// TwinCAT 3 PLC project PLC_UED_SDS
// ProgramVersion: 3.1.4023.0
// libraries:
//   LCLS General, * (SLAC)
//   LCLS Vacuum, * (SLAC - LCLS)
//   lcls-twincat-sample-delivery, * (SLAC)
//   Tc2_Standard, * (Beckhoff Automation GmbH)
//   Tc2_System, * (Beckhoff Automation GmbH)
//   Tc3_Module, * (Beckhoff Automation GmbH)
// project tree:
//   / PlcTask.TcTTO
//   POUs/ MAIN.TcPOU, PRG_RCC.TcPOU
// real-time tasks:
//   TASK PlcTask: cycle T#10ms, priority 20, ADS port 350
// I/O:
//   DEVICE Device 1 (EtherCAT), AmsNetId 172.21.36.53.2.1
//     Term 1 (EK1200) [EK1200-5000 EtherCAT Power supply (2A E-Bus)]
//       RCC_E1 (EL2004)
//       RCC_E2 (EL1004) [EL1004 4Ch. Dig. Input 24V, 3ms]
//       RCC_E3 (EL1004) [EL1004 4Ch. Dig. Input 24V, 3ms]
//       RCC_TC (EL3314) [EL3314 4Ch. Ana. Input Thermocouple (TC)]
//       Term 6 (EK1110) [EK1110 EtherCAT extension]
//     Box 18 (EP9128-0021) [EP9128-0021 8x EtherCAT junction]
//       BR (EP1111-0000) [EP1111-0000 ID-Switch]
//       BR Valves (EP2338-0001) [EP2338-0001 8 Ch. Dig. Input/Output 24V, 0,5A, M8]
//       Term 23 (EP9128-1021) [EP9128-1021 8x EtherCAT junction - Dev A]
//       Term 24 (EP9128-2021) [EP9128-2021 8x EtherCAT junction - Dev B]
//         Box 25 (EP1111) [EP1111-0000 ID-Switch]
//         Box 26 (EP2338-0001) [EP2338-0001 8 Ch. Dig. Input/Output 24V, 0,5A, M8]
//         4PortVICI Serial (EP6002-0002) [EP6002-0002 Interface (RS232/422/485)]
// variable links:
//   PLC_UED_SDS Instance <-> Device 1 (EtherCAT)/Box 18 (EP9128-0021)/BR Valves (EP2338-0001)
//     PlcTask Outputs/MAIN.PURGE_VRC_01_CTL <-> Channel 11/Output
//     PlcTask Outputs/MAIN.PURGE_VRC_02_CTL <-> Channel 12/Output
//     PlcTask Outputs/MAIN.SolenoidPairA.q_xDO1 <-> Channel 9/Output
//     PlcTask Outputs/MAIN.SolenoidPairA.q_xDO2 <-> Channel 10/Output
//   PLC_UED_SDS Instance <-> Device 1 (EtherCAT)/Box 18 (EP9128-0021)/Term 24 (EP9128-2021)/4PortVICI Serial (EP6002-0002)
//     PlcTask Inputs/MAIN.fbValve.fbNporValve.stViciSerial.stComIn/D <-> COM TxPDO-Map Inputs Channel 2/Data In 0
//     PlcTask Inputs/MAIN.fbValve.fbNporValve.stViciSerial.stComIn/D @bit {8..168 step 8} <-> COM TxPDO-Map Inputs Channel 2/Data In {1..21}  (21 links)
//     PlcTask Inputs/MAIN.fbValve.fbNporValve.stViciSerial.stComIn/Status <-> COM TxPDO-Map Inputs Channel 2/Status
//     PlcTask Outputs/MAIN.fbValve.fbNporValve.stViciSerial.stComOut/Ctrl <-> COM RxPDO-Map Outputs Channel 2/Ctrl
//     PlcTask Outputs/MAIN.fbValve.fbNporValve.stViciSerial.stComOut/D <-> COM RxPDO-Map Outputs Channel 2/Data Out 0
//     PlcTask Outputs/MAIN.fbValve.fbNporValve.stViciSerial.stComOut/D @bit {8..168 step 8} <-> COM RxPDO-Map Outputs Channel 2/Data Out {1..21}  (21 links)
//   PLC_UED_SDS Instance <-> Device 1 (EtherCAT)/Term 1 (EK1200)/RCC_E1 (EL2004)
//     PlcTask Outputs/PRG_RCC.RCC_VRC_01.q_xOPN_DO <-> Channel 1/Output
//     PlcTask Outputs/PRG_RCC.RCC_VRC_02.q_xOPN_DO <-> Channel 2/Output
//     PlcTask Outputs/PRG_RCC.RCC_VRC_03.q_xOPN_DO <-> Channel 3/Output
//     PlcTask Outputs/PRG_RCC.RCC_VRC_04.q_xOPN_DO <-> Channel 4/Output
//   PLC_UED_SDS Instance <-> Device 1 (EtherCAT)/Term 1 (EK1200)/RCC_E2 (EL1004)
//     PlcTask Inputs/PRG_RCC.RCC_VRC_01.i_xClsLS <-> Channel 1/Input
//     PlcTask Inputs/PRG_RCC.RCC_VRC_02.i_xClsLS <-> Channel 2/Input
//     PlcTask Inputs/PRG_RCC.RCC_VRC_03.i_xClsLS <-> Channel 3/Input
//     PlcTask Inputs/PRG_RCC.RCC_VRC_04.i_xClsLS <-> Channel 4/Input
//   PLC_UED_SDS Instance <-> Device 1 (EtherCAT)/Term 1 (EK1200)/RCC_GPI (EL3174-0002)
//     PlcTask Inputs/PRG_RCC.RCC_GCP_01.i_iPRESS_R <-> AI Standard Channel 1/Value
//   PLC_UED_SDS Instance <-> Device 1 (EtherCAT)/Term 1 (EK1200)/RCC_TC (EL3314)
//     PlcTask Inputs/PRG_RCC.RCC_STC_01.bError <-> TC Inputs Channel 1/Status/Error
//     PlcTask Inputs/PRG_RCC.RCC_STC_01.bOverrange <-> TC Inputs Channel 1/Status/Overrange
//     PlcTask Inputs/PRG_RCC.RCC_STC_01.bUnderrange <-> TC Inputs Channel 1/Status/Underrange
//     PlcTask Inputs/PRG_RCC.RCC_STC_01.iRaw <-> TC Inputs Channel 1/Value

CONFIGURATION PLC_UED_SDS
    RESOURCE PLC ON TwinCAT3
        TASK PlcTask(INTERVAL := T#10ms, PRIORITY := 20);
        PROGRAM MAIN WITH PlcTask : MAIN;
    END_RESOURCE
END_CONFIGURATION

// ---- POUs/MAIN.TcPOU
PROGRAM MAIN
VAR
    // 4 Port Valve
    {attribute 'pytmc' := 'pv: UED:SDS:VICI:01'}
    {attribute 'TcLinkTo' := '.fbNporValve.stViciSerial.stComIn.Status := TIID^Device 1 (EtherCAT)^Box 18 (EP9128-0021)^Term 24 (EP9128-2021)^4PortVICI Serial (EP6002-0002)^COM TxPDO-Map Inputs Channel 2^Status;
                              .fbNporValve.stViciSerial.stComOut.Ctrl := TIID^Device 1 (EtherCAT)^Box 18 (EP9128-0021)^Term 24 (EP9128-2021)^4PortVICI Serial (EP6002-0002)^COM RxPDO-Map Outputs Channel 2^Ctrl
    '}
    fbValve : FB_4PortViciValve;

    // ON/OFF Valves
    {attribute 'pytmc' := 'pv: UED:SDS:SPR:A'}
    {attribute 'TcLinkTo' := '.q_xDO1 := TIID^Device 1 (EtherCAT)^Box 18 (EP9128-0021)^BR Valves (EP2338-0001)^Channel 9^Output;
                              .q_xDO2 := TIID^Device 1 (EtherCAT)^Box 18 (EP9128-0021)^BR Valves (EP2338-0001)^Channel 10^Output
    '}
    SolenoidPairA : FB_SolenoidPair;

    // Purge Valves
    {attribute 'pytmc' := 'pv: UED:SDS:PURGE:A'}
    {attribute 'TcLinkTo' := 'TIID^Device 1 (EtherCAT)^Box 18 (EP9128-0021)^BR Valves (EP2338-0001)^Channel 11^Output'}
    PURGE_VRC_01_CTL AT%Q* : BOOL;

    {attribute 'pytmc' := 'pv: UED:SDS:PURGE:B'}
    {attribute 'TcLinkTo' := 'TIID^Device 1 (EtherCAT)^Box 18 (EP9128-0021)^BR Valves (EP2338-0001)^Channel 12^Output'}
    PURGE_VRC_02_CTL AT%Q* : BOOL;

END_VAR

PRG_RCC();
SolenoidPairA();
fbValve(iAdress:=1);

END_PROGRAM

// ---- POUs/PRG_RCC.TcPOU
PROGRAM PRG_RCC
VAR
    (* OverrideMode *)
    {attribute 'pytmc' := 'pv: UED:RCC:VAC:OVRD_MODE'}
    xSystemOverrideMode_RCC	: BOOL := FALSE;


    {attribute 'pytmc' :=' pv: UED:RCC:VRC:01 '}
    {attribute 'TcLinkTo' := 	'.i_xClsLS	:=  TIID^Device 1 (EtherCAT)^Term 1 (EK1200)^RCC_E2 (EL1004)^Channel 1^Input;
                                .q_xOPN_DO	:=	TIID^Device 1 (EtherCAT)^Term 1 (EK1200)^RCC_E1 (EL2004)^Channel 1^Output'}
    RCC_VRC_01 : FB_VRC_NC_ClsLS;


    {attribute 'pytmc' :=' pv: UED:RCC:VRC:02 '}
    {attribute 'TcLinkTo' := 	'.i_xClsLS	:=  TIID^Device 1 (EtherCAT)^Term 1 (EK1200)^RCC_E2 (EL1004)^Channel 2^Input;
                                .q_xOPN_DO	:=	TIID^Device 1 (EtherCAT)^Term 1 (EK1200)^RCC_E1 (EL2004)^Channel 2^Output'}
    RCC_VRC_02 : FB_VRC_NC_ClsLS;

    // RIX RCC USES
    //{attribute 'pytmc' :=' pv: UED:RCC:VRC:02 '}
    //{attribute 'TcLinkTo' := 	'.i_xOpnLS	:= 	TIID^Device 1 (EtherCAT)^Term 1 (EK1200)^RCC_E2 (EL1004)^Channel 3^Input;
    //                             .i_xClsLS	:=	TIID^Device 1 (EtherCAT)^Term 1 (EK1200)^RCC_E2 (EL1004)^Channel 4^Input;
    //                            .q_xOPN_DO	:=	TIID^Device 1 (EtherCAT)^Term 1 (EK1200)^RCC_E1 (EL2004)^Channel 2^Output'}
    //RCC_VRC_02 : FB_VRC;

    {attribute 'pytmc' :=' pv: UED:RCC:VRC:03 '}
    {attribute 'TcLinkTo' := 	'.i_xClsLS	:=	TIID^Device 1 (EtherCAT)^Term 1 (EK1200)^RCC_E2 (EL1004)^Channel 3^Input;
                                .q_xOPN_DO	:= 	TIID^Device 1 (EtherCAT)^Term 1 (EK1200)^RCC_E1 (EL2004)^Channel 3^Output'}
    RCC_VRC_03 : FB_VRC_NC_ClsLS;


    {attribute 'pytmc' :=' pv: UED:RCC:VRC:04 '}
    {attribute 'TcLinkTo' := 	'.i_xClsLS	:=	TIID^Device 1 (EtherCAT)^Term 1 (EK1200)^RCC_E2 (EL1004)^Channel 4^Input;
                                .q_xOPN_DO	:=  TIID^Device 1 (EtherCAT)^Term 1 (EK1200)^RCC_E1 (EL2004)^Channel 4^Output'}
    RCC_VRC_04 : FB_VRC_NC_ClsLS;


    {attribute 'pytmc' :=' pv: UED:RCC:GCP:01 '}
    {attribute 'TcLinkTo' := 	'.i_iPRESS_R	:= TIID^Device 1 (EtherCAT)^Term 1 (EK1200)^RCC_GPI (EL3174-0002)^AI Standard Channel 1^Value'}
    RCC_GCP_01 : FB_972;


    {attribute 'pytmc' :=' pv: UED:RCC:TC:01 '}
    {attribute 'TcLinkTo' := ' .bError 		:=	TIID^Device 1 (EtherCAT)^Term 1 (EK1200)^RCC_TC (EL3314)^TC Inputs Channel 1^Status^Error;
                               .bUnderrange :=	TIID^Device 1 (EtherCAT)^Term 1 (EK1200)^RCC_TC (EL3314)^TC Inputs Channel 1^Status^Underrange;
                               .bOverrange 	:=	TIID^Device 1 (EtherCAT)^Term 1 (EK1200)^RCC_TC (EL3314)^TC Inputs Channel 1^Status^Overrange ;
                               .iRaw		:= TIID^Device 1 (EtherCAT)^Term 1 (EK1200)^RCC_TC (EL3314)^TC Inputs Channel 1^Value '}
   RCC_STC_01 : FB_TempSensor;

    RCC_VRC_01_OPEN_OK : BOOL;
    RCC_VRC_02_OPEN_OK : BOOL;
    RCC_VRC_03_OPEN_OK : BOOL;
    RCC_VRC_04_OPEN_OK : BOOL;

   {attribute 'pytmc' :=' pv: UED:GCP:01:INLK_Setpoint '}
    RCC_GCP_01_INTERLOCK_SETPOINT : REAL := 10;

END_VAR

RCC_GCP_01.M_SetBits(30518);
RCC_GCP_01(PG=>);
RCC_STC_01();

(* Valve can open only when UED-RCC-VRC-02 and 03 are closed*)
RCC_VRC_01_OPEN_OK := ( RCC_VRC_02.iq_stValve.i_xClsLS AND NOT RCC_VRC_02.iq_stValve.q_xOPN_DO ) AND
                                    ( RCC_VRC_03.iq_stValve.i_xClsLS AND NOT RCC_VRC_03.iq_stValve.q_xOPN_DO ) ;

RCC_VRC_01(i_xExtILK_OK := RCC_VRC_01_OPEN_OK,
                i_xOverrideMode := xSystemOverrideMode_RCC,
                 iq_stValve=> );

(* Valve can open only when UED-RCC-VRC-01 and 04 are closed*)
RCC_VRC_02_OPEN_OK := ( RCC_VRC_01.iq_stValve.i_xClsLS AND NOT RCC_VRC_01.iq_stValve.q_xOPN_DO ) AND
                                    ( RCC_VRC_04.iq_stValve.i_xClsLS AND NOT RCC_VRC_04.iq_stValve.q_xOPN_DO );

RCC_VRC_02(i_xExtILK_OK := RCC_VRC_02_OPEN_OK,
                i_xOverrideMode := xSystemOverrideMode_RCC,
                 iq_stValve=> );

(* Valve can open only when UED-RCC-GCP-01 reading < setpoint Torr and UED-RCC-VRC-01 and 04 are closed*)
RCC_VRC_03_OPEN_OK := (RCC_GCP_01.PG.rPRESS < RCC_GCP_01_INTERLOCK_SETPOINT and RCC_GCP_01.PG.xPRESS_OK ) AND
                                 ( RCC_VRC_01.iq_stValve.i_xClsLS AND NOT RCC_VRC_01.iq_stValve.q_xOPN_DO ) AND
                                              ( RCC_VRC_04.iq_stValve.i_xClsLS AND NOT RCC_VRC_04.iq_stValve.q_xOPN_DO );

RCC_VRC_03(i_xExtILK_OK := RCC_VRC_03_OPEN_OK,
                i_xOverrideMode := xSystemOverrideMode_RCC,
                 iq_stValve=> );

(* Valve can open only when UED-RCC-VRC-02 and 03 are closed*)
RCC_VRC_04_OPEN_OK := ( RCC_VRC_02.iq_stValve.i_xClsLS AND NOT RCC_VRC_02.iq_stValve.q_xOPN_DO ) AND
                                      ( RCC_VRC_03.iq_stValve.i_xClsLS AND NOT RCC_VRC_03.iq_stValve.q_xOPN_DO ) ;

RCC_VRC_04(i_xExtILK_OK := RCC_VRC_04_OPEN_OK,
                i_xOverrideMode := xSystemOverrideMode_RCC,
                 iq_stValve=> );

END_PROGRAM
